(* IEC 61131-3 sources: AXOpen/src/components.rexroth.tightening/ctrl/src/Axo_CS351_compact (part 2) *)

                    Outputs.CwAnd := FALSE;
                    Outputs.CwLock := TRUE;

                    IF Inputs.CwLockAck THEN
                        THIS.CallTimers(FALSE);
                        _progress := 311;
                    END_IF;
                END_IF;
                // DisableClockwiseTask finished.
                IF _progress = 311 THEN
                    DisableClockwiseTask.DoneWhen(TRUE);
                    _progress := 0;
                END_IF;

                THIS.CallTimers(TRUE);

                DisableClockwiseTask.ThrowWhen(_errorTimer.output);
                Status.Action.Id := TO_UINT(_progress);
                DisableClockwiseTask.ThrowWhen(DisableClockwiseTask.Duration >= Config.TaskTimeout AND Config.TaskTimeout > T#0s ,'<#DisableClockwiseTask timeout.#>');
            END_IF;
            IF DisableClockwiseTask.DoneReached() THEN
                Status.Action.Id :=  UINT#111;
                Status.Error.Id :=  UINT#0;
            ELSIF DisableClockwiseTask.ErrorOccured() THEN
                Status.Action.Id :=  UINT#10010;
                Status.Error.Id  :=  UINT#10010;
            ELSIF DisableClockwiseTask.AbortTriggered()THEN
                Status.Action.Id :=  UINT#10011;
                Status.Error.Id  :=  UINT#10011;
            END_IF;
            Messenger.ActivateOnCondition(ULINT#10010,DisableClockwiseTask.HasError(), eAxoMessageCategory#Error);
            Messenger.ActivateOnCondition(ULINT#10011,DisableClockwiseTask.IsAborted(), eAxoMessageCategory#Error);
            Messenger.ActivateOnCondition(ULINT#112,DisableClockwiseTask.RestoreTriggered() , eAxoMessageCategory#Error);
            IF DisableClockwiseTask.RestoreTriggered() AND _progress >= 310 AND _progress <= 314  THEN
                Status.Action.Id :=  UINT#112;
                _progress := 0;
            END_IF;
            //**************************************************

            //*************EnableClockwiseTask******************
            EnableClockwiseTask.SetIsDisabled(FALSE);
            IF EnableClockwiseTask.StartTriggered() THEN
                Status.Action.Id :=  UINT#115;
            END_IF;
            Messenger.ActivateOnCondition(ULINT#115,EnableClockwiseTask.IsBusy(), eAxoMessageCategory#Info);
            Messenger.ActivateOnCondition(ULINT#116,EnableClockwiseTask.IsDone(), eAxoMessageCategory#Info);
            IF EnableClockwiseTask.Execute(THIS) THEN
                IF _progress = 0 THEN
                    Status.Error.Id := UINT#0;
                    TaskMessenger.Restore();
                    THIS.CallTimers(FALSE);
                    _progress := 315;
                END_IF;
                // EnableClockwiseTask running: waiting for 'Inputs.CwLockAck' to be off.
                IF _progress = 315 THEN
                    IF _infoTimer.output THEN
                        TaskMessenger.Activate( UINT#515, eAxoMessageCategory#Warning);
                        Status.Error.Id :=      UINT#515;
                    END_IF;

                    Outputs.CwAnd := TRUE;
                    Outputs.CwLock := FALSE;

                    IF NOT Inputs.CwLockAck THEN
                        THIS.CallTimers(FALSE);
                        _progress := 316;
                    END_IF;
                END_IF;
                // EnableClockwiseTask finished.
                IF _progress = 316 THEN
                    EnableClockwiseTask.DoneWhen(TRUE);
                    _progress := 0;
                END_IF;

                THIS.CallTimers(TRUE);

                EnableClockwiseTask.ThrowWhen(_errorTimer.output);
                Status.Action.Id := TO_UINT(_progress);
                EnableClockwiseTask.ThrowWhen(EnableClockwiseTask.Duration >= Config.TaskTimeout AND Config.TaskTimeout > T#0s ,'<#EnableClockwiseTask timeout.#>');
            END_IF;
            IF EnableClockwiseTask.DoneReached() THEN
                Status.Action.Id :=  UINT#116;
                Status.Error.Id :=  UINT#0;
            ELSIF EnableClockwiseTask.ErrorOccured() THEN
                Status.Action.Id :=  UINT#10015;
                Status.Error.Id  :=  UINT#10015;
            ELSIF EnableClockwiseTask.AbortTriggered()THEN
                Status.Action.Id :=  UINT#10016;
                Status.Error.Id  :=  UINT#10016;
            END_IF;
            Messenger.ActivateOnCondition(ULINT#10015,EnableClockwiseTask.HasError(), eAxoMessageCategory#Error);
            Messenger.ActivateOnCondition(ULINT#10016,EnableClockwiseTask.IsAborted(), eAxoMessageCategory#Error);
            Messenger.ActivateOnCondition(ULINT#117,EnableClockwiseTask.RestoreTriggered() , eAxoMessageCategory#Error);
            IF EnableClockwiseTask.RestoreTriggered() AND _progress >= 315 AND _progress <= 319  THEN
                Status.Action.Id :=  UINT#117;
                _progress := 0;
            END_IF;
            //**************************************************

            //*************DisableCounterClockwiseTask**********
            DisableCounterClockwiseTask.SetIsDisabled(FALSE);
            IF DisableCounterClockwiseTask.StartTriggered() THEN
                Status.Action.Id :=  UINT#120;
            END_IF;
            Messenger.ActivateOnCondition(ULINT#120,DisableCounterClockwiseTask.IsBusy(), eAxoMessageCategory#Info);
            Messenger.ActivateOnCondition(ULINT#121,DisableCounterClockwiseTask.IsDone(), eAxoMessageCategory#Info);
            IF DisableCounterClockwiseTask.Execute(THIS) THEN
                IF _progress = 0 THEN
                    Status.Error.Id := UINT#0;
                    TaskMessenger.Restore();
                    THIS.CallTimers(FALSE);
                    _progress := 320;
                END_IF;
                // DisableCounterClockwiseTask running: waiting for 'Inputs.CcwLockAck' to be on.
                IF _progress = 320 THEN
                    IF _infoTimer.output THEN
                        TaskMessenger.Activate( UINT#520, eAxoMessageCategory#Warning);
                        Status.Error.Id :=      UINT#520;
                    END_IF;

                    Outputs.CcwAnd := FALSE;
                    Outputs.CcwLock := TRUE;

                    IF Inputs.CcwLockAck THEN
                        THIS.CallTimers(FALSE);
                        _progress := 321;
                    END_IF;
                END_IF;
                // DisableCounterClockwiseTask  finished.
                IF _progress = 321 THEN
                    DisableCounterClockwiseTask.DoneWhen(TRUE);
                    _progress := 0;
                END_IF;

                THIS.CallTimers(TRUE);

                DisableCounterClockwiseTask.ThrowWhen(_errorTimer.output);
                Status.Action.Id := TO_UINT(_progress);
                DisableCounterClockwiseTask.ThrowWhen(DisableCounterClockwiseTask.Duration >= Config.TaskTimeout AND Config.TaskTimeout > T#0s ,'<#DisableCounterClockwiseTask timeout.#>');
            END_IF;
            IF DisableCounterClockwiseTask.DoneReached() THEN
                Status.Action.Id :=  UINT#121;
                Status.Error.Id :=  UINT#0;
            ELSIF DisableCounterClockwiseTask.ErrorOccured() THEN
                Status.Action.Id :=  UINT#10020;
                Status.Error.Id  :=  UINT#10020;
            ELSIF DisableCounterClockwiseTask.AbortTriggered()THEN
                Status.Action.Id :=  UINT#10021;
                Status.Error.Id  :=  UINT#10021;
            END_IF;
            Messenger.ActivateOnCondition(ULINT#10020,DisableCounterClockwiseTask.HasError(), eAxoMessageCategory#Error);
            Messenger.ActivateOnCondition(ULINT#10021,DisableCounterClockwiseTask.IsAborted(), eAxoMessageCategory#Error);
            Messenger.ActivateOnCondition(ULINT#122,DisableCounterClockwiseTask.RestoreTriggered() , eAxoMessageCategory#Error);
            IF DisableCounterClockwiseTask.RestoreTriggered() AND _progress >= 320 AND _progress <= 324  THEN
                Status.Action.Id :=  UINT#122;
                _progress := 0;
            END_IF;
            //**************************************************

            //*************EnableCounterClockwiseTask***********
            EnableCounterClockwiseTask.SetIsDisabled(FALSE);
            IF EnableCounterClockwiseTask.StartTriggered() THEN
                Status.Action.Id :=  UINT#125;
            END_IF;
            Messenger.ActivateOnCondition(ULINT#125,EnableCounterClockwiseTask.IsBusy(), eAxoMessageCategory#Info);
            Messenger.ActivateOnCondition(ULINT#126,EnableCounterClockwiseTask.IsDone(), eAxoMessageCategory#Info);
            IF EnableCounterClockwiseTask.Execute(THIS) THEN
                IF _progress = 0 THEN
                    Status.Error.Id := UINT#0;
                    TaskMessenger.Restore();
                    THIS.CallTimers(FALSE);
                    _progress := 325;
                END_IF;
                // EnableCounterClockwiseTask running: waiting for 'Inputs.CcwLockAck' to be off.
                IF _progress = 325 THEN
                    IF _infoTimer.output THEN
                        TaskMessenger.Activate( UINT#525, eAxoMessageCategory#Warning);
                        Status.Error.Id :=      UINT#525;
                    END_IF;

                    Outputs.CcwAnd := TRUE;
                    Outputs.CcwLock := FALSE;

                    IF NOT Inputs.CcwLockAck THEN
                        THIS.CallTimers(FALSE);
                        _progress := 326;
                    END_IF;
                END_IF;
                // EnableCounterClockwiseTask finished.
                IF _progress = 326 THEN
                    EnableCounterClockwiseTask.DoneWhen(TRUE);
                    _progress := 0;
                END_IF;

                THIS.CallTimers(TRUE);

                EnableCounterClockwiseTask.ThrowWhen(_errorTimer.output);
                Status.Action.Id := TO_UINT(_progress);
                EnableCounterClockwiseTask.ThrowWhen(EnableCounterClockwiseTask.Duration >= Config.TaskTimeout AND Config.TaskTimeout > T#0s ,'<#EnableCounterClockwiseTask timeout.#>');
            END_IF;
            IF EnableCounterClockwiseTask.DoneReached() THEN
                Status.Action.Id :=  UINT#126;
                Status.Error.Id :=  UINT#0;
            ELSIF EnableCounterClockwiseTask.ErrorOccured() THEN
                Status.Action.Id :=  UINT#10025;
                Status.Error.Id  :=  UINT#10025;
            ELSIF EnableCounterClockwiseTask.AbortTriggered()THEN
                Status.Action.Id :=  UINT#10026;
                Status.Error.Id  :=  UINT#10026;
            END_IF;
            Messenger.ActivateOnCondition(ULINT#10025,EnableCounterClockwiseTask.HasError(), eAxoMessageCategory#Error);
            Messenger.ActivateOnCondition(ULINT#10026,EnableCounterClockwiseTask.IsAborted(), eAxoMessageCategory#Error);
            Messenger.ActivateOnCondition(ULINT#127,EnableCounterClockwiseTask.RestoreTriggered() , eAxoMessageCategory#Error);
            IF EnableCounterClockwiseTask.RestoreTriggered() AND _progress >= 325 AND _progress <= 329  THEN
                Status.Action.Id :=  UINT#127;
                _progress := 0;
            END_IF;
            //**************************************************

            //*************ResetFaultTask***********************
            ResetFaultTask.SetIsDisabled(FALSE);
            IF ResetFaultTask.StartTriggered() THEN
                Status.Action.Id :=  UINT#130;
            END_IF;
            Messenger.ActivateOnCondition(ULINT#130,ResetFaultTask.IsBusy(), eAxoMessageCategory#Info);
            Messenger.ActivateOnCondition(ULINT#131,ResetFaultTask.IsDone(), eAxoMessageCategory#Info);
            IF ResetFaultTask.Execute(THIS) THEN
                IF _progress = 0 THEN
                    Status.Error.Id := UINT#0;
                    TaskMessenger.Restore();
                    THIS.CallTimers(FALSE);
                    _progress := 330;
                END_IF;
                // ResetFaultTask running: waiting for 'Inputs.NoFault' to be on.
                IF _progress = 330 THEN
                    IF _infoTimer.output THEN
                        TaskMessenger.Activate( UINT#530, eAxoMessageCategory#Warning);
                        Status.Error.Id :=      UINT#530;
                    END_IF;

                    Outputs.ResetFault := NOT Inputs.NoFault AND _blink.output;

                    IF Inputs.NoFault THEN
                        THIS.CallTimers(FALSE);
                        _progress := 331;
                    END_IF;
                END_IF;
                // ResetFaultTask running: waiting for 'Inputs.Ready' to be on.
                IF _progress = 331 THEN
                    IF _infoTimer.output THEN
                        TaskMessenger.Activate( UINT#531, eAxoMessageCategory#Warning);
                        Status.Error.Id :=      UINT#531;
                    END_IF;

                    IF Inputs.Ready THEN
                        THIS.CallTimers(FALSE);
                        _progress := 332;
                    END_IF;
                END_IF;
                // ResetFaultTask finished.
                IF _progress = 332 THEN
                    ResetFaultTask.DoneWhen(TRUE);
                    _progress := 0;
                END_IF;

                THIS.CallTimers(TRUE);

                ResetFaultTask.ThrowWhen(_errorTimer.output);
                Status.Action.Id := TO_UINT(_progress);
                ResetFaultTask.ThrowWhen(ResetFaultTask.Duration >= Config.TaskTimeout AND Config.TaskTimeout > T#0s ,'<#ResetFaultTask timeout.#>');
            END_IF;
            IF ResetFaultTask.DoneReached() THEN
                Status.Action.Id :=  UINT#131;
                Status.Error.Id :=  UINT#0;
            ELSIF ResetFaultTask.ErrorOccured() THEN
                Status.Action.Id :=  UINT#10030;
                Status.Error.Id  :=  UINT#10030;
            ELSIF ResetFaultTask.AbortTriggered()THEN
                Status.Action.Id :=  UINT#10031;
                Status.Error.Id  :=  UINT#10031;
            END_IF;
            Messenger.ActivateOnCondition(ULINT#10030,ResetFaultTask.HasError(), eAxoMessageCategory#Error);
            Messenger.ActivateOnCondition(ULINT#10031,ResetFaultTask.IsAborted(), eAxoMessageCategory#Error);
            Messenger.ActivateOnCondition(ULINT#132,ResetFaultTask.RestoreTriggered() , eAxoMessageCategory#Error);
            IF ResetFaultTask.RestoreTriggered() AND _progress >= 330 AND _progress <= 334  THEN
                Status.Action.Id :=  UINT#132;
                _progress := 0;
            END_IF;
            //**************************************************

            //*************ResetResultsTask*********************
            ResetResultsTask.SetIsDisabled(FALSE);
            IF ResetResultsTask.StartTriggered() THEN
                Status.Action.Id :=  UINT#135;
            END_IF;
            Messenger.ActivateOnCondition(ULINT#135,ResetResultsTask.IsBusy(), eAxoMessageCategory#Info);
            Messenger.ActivateOnCondition(ULINT#136,ResetResultsTask.IsDone(), eAxoMessageCategory#Info);
            IF ResetResultsTask.Execute(THIS) THEN
                IF _progress = 0 THEN
                    Status.Error.Id := UINT#0;
                    TaskMessenger.Restore();
                    THIS.CallTimers(FALSE);
                    _progress := 335;
                END_IF;
                // ResetResultsTask running: waiting for 'Inputs.CycleComplete' to be off.
                IF _progress = 335 THEN
                    IF _infoTimer.output THEN
                        TaskMessenger.Activate( UINT#535, eAxoMessageCategory#Warning);
                        Status.Error.Id :=      UINT#535;
                    END_IF;

                    Outputs.ResetResults := Inputs.CycleComplete AND _blink.output;
                    IF NOT Inputs.CycleComplete THEN
                        Outputs.ResetResults := FALSE;
                        THIS.CallTimers(FALSE);
                        _progress := 336;
                    END_IF;
                END_IF;
                // ResetResultsTask finished.
                IF _progress = 336 THEN
                    ResetResultsTask.DoneWhen(TRUE);
                    _progress := 0;
                END_IF;

                THIS.CallTimers(TRUE);

                ResetResultsTask.ThrowWhen(_errorTimer.output);
                Status.Action.Id := TO_UINT(_progress);
                ResetResultsTask.ThrowWhen(ResetResultsTask.Duration >= Config.TaskTimeout AND Config.TaskTimeout > T#0s ,'<#ResetResultsTask timeout.#>');
            END_IF;
            IF ResetResultsTask.DoneReached() THEN
                Status.Action.Id :=  UINT#136;
                Status.Error.Id :=  UINT#0;
            ELSIF ResetResultsTask.ErrorOccured() THEN
                Status.Action.Id :=  UINT#10035;
                Status.Error.Id  :=  UINT#10035;
            ELSIF ResetResultsTask.AbortTriggered()THEN
                Status.Action.Id :=  UINT#10036;
                Status.Error.Id  :=  UINT#10036;
            END_IF;
            Messenger.ActivateOnCondition(ULINT#10035,ResetResultsTask.HasError(), eAxoMessageCategory#Error);
            Messenger.ActivateOnCondition(ULINT#10036,ResetResultsTask.IsAborted(), eAxoMessageCategory#Error);
            Messenger.ActivateOnCondition(ULINT#137,ResetResultsTask.RestoreTriggered() , eAxoMessageCategory#Error);
            IF ResetResultsTask.RestoreTriggered() AND _progress >= 335 AND _progress <= 339  THEN
                Status.Action.Id :=  UINT#137;
                _progress := 0;
            END_IF;
            //**************************************************

            //*************SetScrewingProgramTask***************
            SetScrewingProgramTask.SetIsDisabled(FALSE);
            IF SetScrewingProgramTask.StartTriggered() THEN
                Status.Action.Id :=  UINT#140;
            END_IF;
            Messenger.ActivateOnCondition(ULINT#140,SetScrewingProgramTask.IsBusy(), eAxoMessageCategory#Info);
            Messenger.ActivateOnCondition(ULINT#141,SetScrewingProgramTask.IsDone(), eAxoMessageCategory#Info);
            IF SetScrewingProgramTask.Execute(THIS) THEN
                IF _progress = 0 THEN
                    Status.Error.Id := UINT#0;
                    TaskMessenger.Restore();
                    THIS.CallTimers(FALSE);
                    _progress := 340;
                END_IF;
                // SetScrewingProgramTask running: checking actual screwing program number.
                IF _progress = 340 THEN
                    IF _infoTimer.output THEN
                        TaskMessenger.Activate( UINT#540, eAxoMessageCategory#Warning);
                        Status.Error.Id :=      UINT#540;
                    END_IF;

                    IF _programNo <> Inputs.ProgramNo THEN
                        THIS.CallTimers(FALSE);
                        _progress := 341;
                    ELSE
                        THIS.CallTimers(FALSE);
                        _progress := 344;
                    END_IF;
                END_IF;
                // SetScrewingProgramTask running: checking required screwing program number.
                IF _progress = 341 THEN
                    IF _infoTimer.output THEN
                        TaskMessenger.Activate( UINT#541, eAxoMessageCategory#Warning);
                        Status.Error.Id :=      UINT#541;
                    END_IF;

                    IF _programNo>=BYTE#0 AND _programNo<=BYTE#99 THEN
                        THIS.CallTimers(FALSE);
                        _progress := 342;
                    ELSE
                        Messenger.Activate(ULINT#2000,eAxoMessageCategory#ProgrammingError);
                    END_IF;
                END_IF;
                // SetScrewingProgramTask running: waiting for 'Inputs.Ready' to be on.
                IF _progress = 342 THEN
                    IF _infoTimer.output THEN
                        TaskMessenger.Activate( UINT#542, eAxoMessageCategory#Warning);
                        Status.Error.Id :=      UINT#542;
                    END_IF;

                    IF Inputs.Ready THEN
                        THIS.CallTimers(FALSE);
                        _progress := 343;
                    END_IF;
                END_IF;
                // SetScrewingProgramTask running: waiting for the program to be set.
                IF _progress = 343 THEN
                    IF _infoTimer.output THEN
                        TaskMessenger.Activate( UINT#543, eAxoMessageCategory#Warning);
                        Status.Error.Id :=      UINT#543;
                    END_IF;

                    Outputs.ProgramNo := _programNo;

                    IF Inputs.ProgramNoAck = Outputs.ProgramNo THEN
                        THIS.CallTimers(FALSE);
                        _progress := 344;
                    END_IF;
                END_IF;
                // SetScrewingProgramTask finished.
                IF _progress = 344 THEN
                    SetScrewingProgramTask.DoneWhen(TRUE);
                    _progress := 0;
                END_IF;

                THIS.CallTimers(TRUE);

                SetScrewingProgramTask.ThrowWhen(_errorTimer.output);
                Status.Action.Id := TO_UINT(_progress);
                SetScrewingProgramTask.ThrowWhen(SetScrewingProgramTask.Duration >= Config.TaskTimeout AND Config.TaskTimeout > T#0s ,'<#SetScrewingProgramTask timeout.#>');
            END_IF;
            IF SetScrewingProgramTask.DoneReached() THEN
                Status.Action.Id :=  UINT#141;
                Status.Error.Id :=  UINT#0;
            ELSIF SetScrewingProgramTask.ErrorOccured() THEN
                Status.Action.Id :=  UINT#10040;
                Status.Error.Id  :=  UINT#10040;
            ELSIF SetScrewingProgramTask.AbortTriggered()THEN
                Status.Action.Id :=  UINT#10041;
                Status.Error.Id  :=  UINT#10041;
            END_IF;
            Messenger.ActivateOnCondition(ULINT#10040,SetScrewingProgramTask.HasError(), eAxoMessageCategory#Error);
            Messenger.ActivateOnCondition(ULINT#10041,SetScrewingProgramTask.IsAborted(), eAxoMessageCategory#Error);
            Messenger.ActivateOnCondition(ULINT#142,SetScrewingProgramTask.RestoreTriggered() , eAxoMessageCategory#Error);
            IF SetScrewingProgramTask.RestoreTriggered() AND _progress >= 340 AND _progress <= 344  THEN
                Status.Action.Id :=  UINT#142;
                _progress := 0;
            END_IF;
            //**************************************************

            //*************GetScrewingResultsTask*******************
            GetScrewingResultsTask.SetIsDisabled(FALSE);
            IF GetScrewingResultsTask.StartTriggered() THEN
                Status.Action.Id :=  UINT#150;
            END_IF;
            Messenger.ActivateOnCondition(ULINT#150,GetScrewingResultsTask.IsBusy(), eAxoMessageCategory#Info);
            Messenger.ActivateOnCondition(ULINT#151,GetScrewingResultsTask.IsDone(), eAxoMessageCategory#Info);
            IF GetScrewingResultsTask.Execute(THIS) THEN
                IF _progress = 0 THEN
                    Status.Error.Id := UINT#0;
                    TaskMessenger.Restore();
                    THIS.CallTimers(FALSE);
                    _progress := 350;
                END_IF;
                // GetScrewingResultsTask running.
                IF _progress = 350 THEN
                    IF _infoTimer.output THEN
                        TaskMessenger.Activate( UINT#550, eAxoMessageCategory#Warning);
                        Status.Error.Id :=      UINT#550;
                    END_IF;

                    Results.Result := Inputs.Result;
                    Results.IDcode.Data := Inputs.IDcode;
                    Results.CnoSE := Inputs.CnoSE;
                    Results.ProgramNo := Inputs.ProgramNo;
                    Results.TorqueMin := Inputs.TorqueMin;
                    Results.Torque := Inputs.Torque;
                    Results.TorqueMax := Inputs.TorqueMax;
                    Results.AngleMin := Inputs.AngleMin;
                    Results.Angle := Inputs.Angle;
                    Results.AngleMax := Inputs.AngleMax;
                    Results.ErrorCode := Inputs.ErrorCode;
                    Results.ErrorClass := Inputs.ErrorClass;

                    Results.IDcode.ToggleDataChangedFlag();

                    IF TRUE THEN
                        THIS.CallTimers(FALSE);
                        _progress := 351;
                    END_IF;
                END_IF;
                // GetScrewingResultsTask finished.
                IF _progress = 351 THEN
                    GetScrewingResultsTask.DoneWhen(TRUE);
                    _progress := 0;
                END_IF;

                THIS.CallTimers(TRUE);

                GetScrewingResultsTask.ThrowWhen(_errorTimer.output);
                Status.Action.Id := TO_UINT(_progress);
                GetScrewingResultsTask.ThrowWhen(GetScrewingResultsTask.Duration >= Config.TaskTimeout AND Config.TaskTimeout > T#0s ,'<#GetScrewingResultsTask timeout.#>');
            END_IF;
            IF GetScrewingResultsTask.DoneReached() THEN
                Status.Action.Id :=  UINT#151;
                Status.Error.Id :=  UINT#0;
            ELSIF GetScrewingResultsTask.ErrorOccured() THEN
                Status.Action.Id :=  UINT#10050;
                Status.Error.Id  :=  UINT#10050;
            ELSIF GetScrewingResultsTask.AbortTriggered()THEN
                Status.Action.Id :=  UINT#10051;
                Status.Error.Id  :=  UINT#10051;
            END_IF;
            Messenger.ActivateOnCondition(ULINT#10050,GetScrewingResultsTask.HasError(), eAxoMessageCategory#Error);
            Messenger.ActivateOnCondition(ULINT#10051,GetScrewingResultsTask.IsAborted(), eAxoMessageCategory#Error);
            Messenger.ActivateOnCondition(ULINT#152,GetScrewingResultsTask.RestoreTriggered() , eAxoMessageCategory#Error);
            IF GetScrewingResultsTask.RestoreTriggered() AND _progress >= 350 AND _progress <= 359  THEN
                Status.Action.Id :=  UINT#152;
                _progress := 0;
            END_IF;
            //**************************************************

            //*************ScrewClockwiseTask*******************
            ScrewClockwiseTask.SetIsDisabled(FALSE);
            IF ScrewClockwiseTask.StartTriggered() THEN
                Status.Action.Id :=  UINT#160;
            END_IF;
            Messenger.ActivateOnCondition(ULINT#160,ScrewClockwiseTask.IsBusy(), eAxoMessageCategory#Info);
            Messenger.ActivateOnCondition(ULINT#161,ScrewClockwiseTask.IsDone(), eAxoMessageCategory#Info);
            IF ScrewClockwiseTask.Execute(THIS) THEN
                IF _progress = 0 THEN
                    Status.Error.Id := UINT#0;
                    TaskMessenger.Restore();
                    THIS.CallTimers(FALSE);
                    _progress := 360;
                END_IF;
                // ScrewClockwiseTask running: waiting for 'Inputs.Ready' to be on.
                IF _progress = 360 THEN
                    IF _infoTimer.output THEN
                        TaskMessenger.Activate( UINT#560, eAxoMessageCategory#Warning);
                        Status.Error.Id :=      UINT#560;
                    END_IF;

                    IF Inputs.Ready THEN
                        THIS.CallTimers(FALSE);
                        _progress := 361;
                    END_IF;
                END_IF;
                // ScrewClockwiseTask running: waiting for 'Inputs.EnableAck' to be on.
                IF _progress = 361 THEN
                    IF _infoTimer.output THEN
                        TaskMessenger.Activate( UINT#561, eAxoMessageCategory#Warning);
                        Status.Error.Id :=      UINT#561;
                    END_IF;

                    Outputs.Enable := TRUE;
                    Outputs.ActiveEnable := TRUE;
                    IF Inputs.EnableAck THEN
                        THIS.CallTimers(FALSE);
                        _progress := 362;
                    END_IF;
                END_IF;
                // ScrewClockwiseTask running: waiting for 'Inputs.ActiveEnableAck' to be on.
                IF _progress = 362 THEN
                    IF _infoTimer.output THEN
                        TaskMessenger.Activate( UINT#562, eAxoMessageCategory#Warning);
                        Status.Error.Id :=      UINT#562;
                    END_IF;

                    Outputs.Enable := TRUE;
                    Outputs.ActiveEnable := TRUE;

                    IF Inputs.ActiveEnableAck THEN
                        THIS.CallTimers(FALSE);
                        _progress := 363;
                    END_IF;
                END_IF;
                // ScrewClockwiseTask running: waiting for 'Inputs.CwLockAck' to be off.
                IF _progress = 363 THEN
                    IF _infoTimer.output THEN
                        TaskMessenger.Activate( UINT#563, eAxoMessageCategory#Warning);
                        Status.Error.Id :=      UINT#563;
                    END_IF;

                    Outputs.CwAnd := TRUE;
                    Outputs.CwLock := FALSE;

                    IF NOT Inputs.CwLockAck THEN
                        THIS.CallTimers(FALSE);
                        _progress := 364;
                    END_IF;
                END_IF;
                // ScrewClockwiseTask running: waiting for 'Inputs.InCycle' to be on.
                IF _progress = 364 THEN
                    IF _infoTimer.output THEN
                        TaskMessenger.Activate( UINT#564, eAxoMessageCategory#Warning);
                        Status.Error.Id :=      UINT#564;
                    END_IF;

                    Outputs.StartClockwise := TRUE;

                    IF Inputs.InCycle THEN
                        THIS.CallTimers(FALSE);
                        _progress := 365;
                    END_IF;
                END_IF;
                // ScrewClockwiseTask running: waiting for 'Inputs.InCycle' to be on.
                IF _progress = 365 THEN
                    IF _infoTimer.output THEN
                        TaskMessenger.Activate( UINT#565, eAxoMessageCategory#Warning);
                        Status.Error.Id :=      UINT#565;
                    END_IF;

                    Outputs.StartClockwise := _automaticStart;

                    IF Inputs.InCycle THEN
                        THIS.CallTimers(FALSE);
                        _progress := 366;
                    END_IF;
                END_IF;
                // ScrewClockwiseTask running: waiting for 'Inputs.CycleComplete' to be on.
                IF _progress = 366 THEN
                    IF _infoTimer.output THEN
                        TaskMessenger.Activate( UINT#566, eAxoMessageCategory#Warning);
                        Status.Error.Id :=      UINT#566;
                    END_IF;

                    Outputs.StartClockwise := _automaticStart;

                    IF Inputs.CycleComplete THEN
                        THIS.CallTimers(FALSE);
                        _progress := 367;
                    END_IF;
                END_IF;
                // ScrewClockwiseTask running: waiting for 'Inputs.InCycle' to be off.
                IF _progress = 367 THEN
                    IF _infoTimer.output THEN
                        TaskMessenger.Activate( UINT#567, eAxoMessageCategory#Warning);
                        Status.Error.Id :=      UINT#567;
                    END_IF;

                    Outputs.StartClockwise := FALSE;
                    Outputs.ActiveEnable := FALSE;

                    IF NOT Inputs.InCycle THEN
                        THIS.CallTimers(FALSE);
                        _progress := 368;
                    END_IF;
                END_IF;
                // ScrewClockwiseTask running: waiting for 'Inputs.ActiveEnableAck' to be off.
                IF _progress = 368 THEN
                    IF _infoTimer.output THEN
                        TaskMessenger.Activate( UINT#568, eAxoMessageCategory#Warning);
                        Status.Error.Id :=      UINT#568;
                    END_IF;

                    Outputs.StartClockwise := FALSE;
                    Outputs.ActiveEnable := FALSE;

                    IF NOT Inputs.ActiveEnableAck THEN
                        THIS.CallTimers(FALSE);
                        _progress := 369;
                    END_IF;
                END_IF;
                // ScrewClockwiseTask running: waiting for 'Inputs.CycleComplete' to be on.
                IF _progress = 369 THEN
                    IF _infoTimer.output THEN
                        TaskMessenger.Activate( UINT#569, eAxoMessageCategory#Warning);
                        Status.Error.Id :=      UINT#569;
                    END_IF;

                    Outputs.StartClockwise := FALSE;
                    Outputs.ActiveEnable := FALSE;

                    IF Inputs.CycleComplete THEN
                        THIS.CallTimers(FALSE);
                        _progress := 370;
                    END_IF;
                END_IF;
                // ScrewClockwiseTask running: waiting for 'Inputs.CwLockAck' to be on.
                IF _progress = 370 THEN
                    IF _infoTimer.output THEN
                        TaskMessenger.Activate( UINT#570, eAxoMessageCategory#Warning);
                        Status.Error.Id :=      UINT#570;
                    END_IF;

                    Outputs.CwAnd := FALSE;
                    Outputs.CwLock := TRUE;

                    IF Inputs.CwLockAck THEN
                        THIS.CallTimers(FALSE);
                        _progress := 371;
                    END_IF;
                END_IF;
                // ScrewClockwiseTask running: waiting for 'Inputs.CcwLockAck' to be on.
                IF _progress = 371 THEN
                    IF _infoTimer.output THEN
                        TaskMessenger.Activate( UINT#571, eAxoMessageCategory#Warning);
                        Status.Error.Id :=      UINT#571;
                    END_IF;

                    Outputs.CcwAnd := FALSE;
                    Outputs.CcwLock := TRUE;

                   IF Inputs.CcwLockAck THEN
                        THIS.CallTimers(FALSE);
                        _progress := 372;
                    END_IF;
                END_IF;
                // ScrewClockwiseTask finished.
                IF _progress = 372 THEN
                    ScrewClockwiseTask.DoneWhen(TRUE);
                    _progress := 0;
                END_IF;

                THIS.CallTimers(TRUE);

                ScrewClockwiseTask.ThrowWhen(_errorTimer.output);
                Status.Action.Id := TO_UINT(_progress);
                ScrewClockwiseTask.ThrowWhen(ScrewClockwiseTask.Duration >= Config.TaskTimeout AND Config.TaskTimeout > T#0s ,'<#ScrewClockwiseTask timeout.#>');
            END_IF;
            IF ScrewClockwiseTask.DoneReached() THEN
                Status.Action.Id :=  UINT#161;
                Status.Error.Id :=  UINT#0;
            ELSIF ScrewClockwiseTask.ErrorOccured() THEN
                Status.Action.Id :=  UINT#10060;
                Status.Error.Id  :=  UINT#10060;
            ELSIF ScrewClockwiseTask.AbortTriggered()THEN
                Status.Action.Id :=  UINT#10061;
                Status.Error.Id  :=  UINT#10061;
            END_IF;
            Messenger.ActivateOnCondition(ULINT#10060,ScrewClockwiseTask.HasError(), eAxoMessageCategory#Error);
            Messenger.ActivateOnCondition(ULINT#10061,ScrewClockwiseTask.IsAborted(), eAxoMessageCategory#Error);
            Messenger.ActivateOnCondition(ULINT#162,ScrewClockwiseTask.RestoreTriggered() , eAxoMessageCategory#Error);
            IF ScrewClockwiseTask.RestoreTriggered() AND _progress >= 360 AND _progress <= 379  THEN
                Status.Action.Id :=  UINT#162;
                _progress := 0;
            END_IF;
            //*****************************************************

            //*************ScrewCounterClockwiseTask***************
            ScrewCounterClockwiseTask.SetIsDisabled(FALSE);
            IF ScrewCounterClockwiseTask.StartTriggered() THEN
                Status.Action.Id :=  UINT#180;
            END_IF;
            Messenger.ActivateOnCondition(ULINT#180,ScrewCounterClockwiseTask.IsBusy(), eAxoMessageCategory#Info);
            Messenger.ActivateOnCondition(ULINT#181,ScrewCounterClockwiseTask.IsDone(), eAxoMessageCategory#Info);
            IF ScrewCounterClockwiseTask.Execute(THIS) THEN
                IF _progress = 0 THEN
                    Status.Error.Id := UINT#0;
                    TaskMessenger.Restore();
                    THIS.CallTimers(FALSE);
                    _progress := 380;
                END_IF;
                // ScrewCounterClockwiseTask running: waiting for 'Inputs.Ready' to be on.
                IF _progress = 380 THEN
                    IF _infoTimer.output THEN
                        TaskMessenger.Activate( UINT#580, eAxoMessageCategory#Warning);
                        Status.Error.Id :=      UINT#580;
                    END_IF;

                    IF Inputs.Ready THEN
                        THIS.CallTimers(FALSE);
                        _progress := 381;
                    END_IF;
                END_IF;
                // ScrewCounterClockwiseTask running: waiting for 'Inputs.EnableAck' to be on.
                IF _progress = 381 THEN
                    IF _infoTimer.output THEN
                        TaskMessenger.Activate( UINT#581, eAxoMessageCategory#Warning);
                        Status.Error.Id :=      UINT#581;
                    END_IF;

                    Outputs.Enable := TRUE;
                    Outputs.ActiveEnable := TRUE;
                    IF Inputs.EnableAck THEN
                        THIS.CallTimers(FALSE);
                        _progress := 382;
                    END_IF;
                END_IF;
                // ScrewCounterClockwiseTask running: waiting for 'Inputs.ActiveEnableAck' to be on.
                IF _progress = 382 THEN
                    IF _infoTimer.output THEN
                        TaskMessenger.Activate( UINT#582, eAxoMessageCategory#Warning);
                        Status.Error.Id :=      UINT#582;
                    END_IF;

                    Outputs.Enable := TRUE;
                    Outputs.ActiveEnable := TRUE;
                    IF Inputs.ActiveEnableAck THEN
                        THIS.CallTimers(FALSE);
                        _progress := 383;
                    END_IF;
                END_IF;
                // ScrewCounterClockwiseTask running: waiting for 'Inputs.CcwLockAck' to be off.
                IF _progress = 383 THEN
                    IF _infoTimer.output THEN
                        TaskMessenger.Activate( UINT#583, eAxoMessageCategory#Warning);
                        Status.Error.Id :=      UINT#583;
                    END_IF;

                    Outputs.CcwAnd := TRUE;
                    Outputs.CcwLock := FALSE;
                    IF NOT Inputs.CcwLockAck THEN
                        THIS.CallTimers(FALSE);
                        _progress := 384;
                    END_IF;
                END_IF;
                // ScrewCounterClockwiseTask running: waiting for 'Inputs.InCycleCcw' to be on.
                IF _progress = 384 THEN
                    IF _infoTimer.output THEN
                        TaskMessenger.Activate( UINT#584, eAxoMessageCategory#Warning);
                        Status.Error.Id :=      UINT#584;
                    END_IF;

                    IF _automaticStart THEN
                        Outputs.StartCounterClockwise := TRUE;
                    END_IF;
                    IF Inputs.InCycleCcw THEN
                        THIS.CallTimers(FALSE);
                        _progress := 385;
                    END_IF;
                END_IF;
                // ScrewCounterClockwiseTask running: waiting for 'Inputs.InCycleCcw' to be on.
                IF _progress = 385 THEN
                    IF _infoTimer.output THEN
                        TaskMessenger.Activate( UINT#585, eAxoMessageCategory#Warning);
                        Status.Error.Id :=      UINT#585;
                    END_IF;

                    Outputs.StartCounterClockwise := TRUE;
                    IF Inputs.InCycleCcw THEN
                        THIS.CallTimers(FALSE);
                        _progress := 386;
                    END_IF;
                END_IF;
                // ScrewCounterClockwiseTask running: waiting for 'Inputs.CycleComplete' to be on.
                IF _progress = 386 THEN
                    IF _infoTimer.output THEN
                        TaskMessenger.Activate( UINT#586, eAxoMessageCategory#Warning);
                        Status.Error.Id :=      UINT#586;
                    END_IF;

                    Outputs.StartCounterClockwise := TRUE;
                    IF Inputs.CycleComplete THEN
                        THIS.CallTimers(FALSE);
                        _progress := 387;
                    END_IF;
                END_IF;
                // ScrewCounterClockwiseTask running: waiting for 'Inputs.InCycleCcw' to be off.
                IF _progress = 387 THEN
                    IF _infoTimer.output THEN
                        TaskMessenger.Activate( UINT#587, eAxoMessageCategory#Warning);
                        Status.Error.Id :=      UINT#587;
                    END_IF;

                    Outputs.StartCounterClockwise := FALSE;
                    Outputs.ActiveEnable := FALSE;

                    IF NOT Inputs.InCycleCcw THEN
                        THIS.CallTimers(FALSE);
                        _progress := 388;
                    END_IF;
                END_IF;
                // ScrewCounterClockwiseTask running: waiting for 'Inputs.ActiveEnableAck' to be off.
                IF _progress = 388 THEN
                    IF _infoTimer.output THEN
                        TaskMessenger.Activate( UINT#588, eAxoMessageCategory#Warning);
                        Status.Error.Id :=      UINT#588;
                    END_IF;

                    Outputs.StartCounterClockwise := FALSE;
                    Outputs.ActiveEnable := FALSE;

                    IF NOT Inputs.ActiveEnableAck THEN
                        THIS.CallTimers(FALSE);
                        _progress := 389;
                    END_IF;
                END_IF;
                // ScrewCounterClockwiseTask running: waiting for 'Inputs.CycleComplete' to be on.
                IF _progress = 389 THEN
                    IF _infoTimer.output THEN
                        TaskMessenger.Activate( UINT#589, eAxoMessageCategory#Warning);
                        Status.Error.Id :=      UINT#589;
                    END_IF;

                    Outputs.StartCounterClockwise := FALSE;
                    Outputs.ActiveEnable := FALSE;

                    IF Inputs.CycleComplete THEN
                        THIS.CallTimers(FALSE);
                        _progress := 390;
                    END_IF;
                END_IF;
                // ScrewCounterClockwiseTask running: waiting for 'Inputs.CcwLockAck' to be on.
                IF _progress = 390 THEN
                    IF _infoTimer.output THEN
                        TaskMessenger.Activate( UINT#590, eAxoMessageCategory#Warning);
                        Status.Error.Id :=      UINT#590;
                    END_IF;

                    Outputs.CcwAnd := FALSE;
                    Outputs.CcwLock := TRUE;
                    IF Inputs.CcwLockAck THEN
                        THIS.CallTimers(FALSE);
                        _progress := 391;
                    END_IF;
                END_IF;
                // ScrewCounterClockwiseTask running: waiting for 'Inputs.CwLockAck' to be on.
                IF _progress = 391 THEN
                    IF _infoTimer.output THEN
                        TaskMessenger.Activate( UINT#591, eAxoMessageCategory#Warning);
                        Status.Error.Id :=      UINT#591;
                    END_IF;

                    Outputs.CwAnd := FALSE;
                    Outputs.CwLock := TRUE;
                    IF Inputs.CwLockAck THEN
                        THIS.CallTimers(FALSE);
                        _progress := 392;
                    END_IF;
                END_IF;
                // ScrewCounterClockwiseTask finished.
                IF _progress = 392 THEN
                    ScrewCounterClockwiseTask.DoneWhen(TRUE);
                    _progress := 0;
                END_IF;

                THIS.CallTimers(TRUE);

                ScrewCounterClockwiseTask.ThrowWhen(_errorTimer.output);
                Status.Action.Id := TO_UINT(_progress);
                ScrewCounterClockwiseTask.ThrowWhen(ScrewCounterClockwiseTask.Duration >= Config.TaskTimeout AND Config.TaskTimeout > T#0s ,'<#ScrewCounterClockwiseTask timeout.#>');
            END_IF;
            IF ScrewCounterClockwiseTask.DoneReached() THEN
                Status.Action.Id :=  UINT#181;
                Status.Error.Id :=  UINT#0;
            ELSIF ScrewCounterClockwiseTask.ErrorOccured() THEN
                Status.Action.Id :=  UINT#10080;
                Status.Error.Id  :=  UINT#10080;
            ELSIF ScrewCounterClockwiseTask.AbortTriggered()THEN
                Status.Action.Id :=  UINT#10081;
                Status.Error.Id  :=  UINT#10081;
            END_IF;
            Messenger.ActivateOnCondition(ULINT#10080,ScrewCounterClockwiseTask.HasError(), eAxoMessageCategory#Error);
            Messenger.ActivateOnCondition(ULINT#10081,ScrewCounterClockwiseTask.IsAborted(), eAxoMessageCategory#Error);
            Messenger.ActivateOnCondition(ULINT#182,ScrewCounterClockwiseTask.RestoreTriggered() , eAxoMessageCategory#Error);
            IF ScrewCounterClockwiseTask.RestoreTriggered() AND _progress >= 380 AND _progress <= 399  THEN
                Status.Action.Id :=  UINT#182;
                _progress := 0;
            END_IF;
            //**************************************************

            //*************RunAutomatTask***********************
            RunAutomatTask.SetIsDisabled(FALSE);
            IF RunAutomatTask.StartTriggered() THEN
                Status.Action.Id :=  UINT#200;
            END_IF;
            Messenger.ActivateOnCondition(ULINT#200,RunAutomatTask.IsBusy(), eAxoMessageCategory#Info);
            Messenger.ActivateOnCondition(ULINT#201,RunAutomatTask.IsDone(), eAxoMessageCategory#Info);
            IF RunAutomatTask.Execute(THIS) THEN
                IF _progress = 0 THEN
                    Status.Error.Id := UINT#0;
                    TaskMessenger.Restore();
                    THIS.CallTimers(FALSE);
                    _progress := 400;
                END_IF;
                // RunAutomatTask running: setting ID code.
                IF _progress = 400 THEN
                    IF _infoTimer.output THEN
                        TaskMessenger.Activate( UINT#600, eAxoMessageCategory#Warning);
                        Status.Error.Id :=      UINT#600;
                    END_IF;

                    OK := FALSE;
                    NOK := FALSE;

                    Outputs.IDcode := _IDcode;

                    IF TRUE THEN
                        THIS.CallTimers(FALSE);
                        _progress := 401;
                    END_IF;
                END_IF;
                // RunAutomatTask running: waiting for 'Inputs.NoFault' to be on.
                IF _progress = 401 THEN
                    IF _infoTimer.output THEN
                        TaskMessenger.Activate( UINT#601, eAxoMessageCategory#Warning);
                        Status.Error.Id :=      UINT#601;
                    END_IF;

                    Outputs.ResetFault := NOT Inputs.NoFault AND _blink.output;
                    IF Inputs.NoFault THEN
                        Outputs.ResetFault := FALSE;
                        THIS.CallTimers(FALSE);
                        _progress := 402;
                    END_IF;
                END_IF;
                // RunAutomatTask running: waiting for 'Inputs.Ready' to be on.
                IF _progress = 402 THEN
                    IF _infoTimer.output THEN
                        TaskMessenger.Activate( UINT#602, eAxoMessageCategory#Warning);
                        Status.Error.Id :=      UINT#602;
                    END_IF;

                    Outputs.ResetFault := NOT Inputs.NoFault AND _blink.output;
                    IF Inputs.Ready THEN
                        Outputs.ResetFault := FALSE;
                        THIS.CallTimers(FALSE);
                        _progress := 403;
                    END_IF;
                END_IF;
                // RunAutomatTask running: checking the actual screwing program number.
                IF _progress = 403 THEN
                    IF _infoTimer.output THEN
                        TaskMessenger.Activate( UINT#603, eAxoMessageCategory#Warning);
                        Status.Error.Id :=      UINT#603;
                    END_IF;

                    IF _programNo <> Inputs.ProgramNo THEN
                        THIS.CallTimers(FALSE);
                        _progress := 404;
                    ELSE
                        THIS.CallTimers(FALSE);
                        _progress := 407;
                    END_IF;
                END_IF;
                // RunAutomatTask running: checking the required screwing program number
                IF _progress = 404 THEN
                    IF _infoTimer.output THEN
                        TaskMessenger.Activate( UINT#604, eAxoMessageCategory#Warning);
                        Status.Error.Id :=      UINT#604;
                    END_IF;

                    IF _programNo>=BYTE#0 AND _programNo<=BYTE#99 THEN
                        THIS.CallTimers(FALSE);
                        _progress := 405;
                    ELSE
                        Messenger.Activate(ULINT#1100,eAxoMessageCategory#ProgrammingError);
                    END_IF;
                END_IF;
                // RunAutomatTask running: waiting for 'Inputs.Ready' to be on.
                IF _progress = 405 THEN
                    IF _infoTimer.output THEN
                        TaskMessenger.Activate( UINT#605, eAxoMessageCategory#Warning);
                        Status.Error.Id :=      UINT#605;
                    END_IF;

                    IF Inputs.Ready THEN
                        THIS.CallTimers(FALSE);
                        _progress := 406;
                    END_IF;
                END_IF;
                // RunAutomatTask running: waiting for the screwing program to be set.
                IF _progress = 406 THEN
                    IF _infoTimer.output THEN
                        TaskMessenger.Activate( UINT#606, eAxoMessageCategory#Warning);
                        Status.Error.Id :=      UINT#606;
                    END_IF;

                    Outputs.ProgramNo := _programNo;

                    IF Inputs.ProgramNoAck = Outputs.ProgramNo THEN
                        THIS.CallTimers(FALSE);
                        _progress := 407;
                    END_IF;
                END_IF;
                // RunAutomatTask running: waiting for 'Inputs.EnableAck' to be on.
                IF _progress = 407 THEN
                    IF _infoTimer.output THEN
                        TaskMessenger.Activate( UINT#607, eAxoMessageCategory#Warning);
                        Status.Error.Id :=      UINT#607;
                    END_IF;

                    Outputs.Enable := TRUE;

                    IF Inputs.EnableAck THEN
                        THIS.CallTimers(FALSE);
                        _progress := 408;
                    END_IF;
                END_IF;
                // RunAutomatTask running: waiting for 'Inputs.CycleComplete' to be off.
                IF _progress = 408 THEN
                    IF _infoTimer.output THEN
                        TaskMessenger.Activate( UINT#608, eAxoMessageCategory#Warning);
                        Status.Error.Id :=      UINT#608;
                    END_IF;

                    Outputs.ResetResults := Inputs.CycleComplete AND _blink.output;
                    IF NOT Inputs.CycleComplete THEN
                        Outputs.ResetResults := FALSE;
                        THIS.CallTimers(FALSE);
                        _progress := 409;
                    END_IF;
                END_IF;
                // RunAutomatTask running: waiting for 'Inputs.ActiveEnableAck' to be on.
                IF _progress = 409 THEN
                    IF _infoTimer.output THEN
                        TaskMessenger.Activate( UINT#609, eAxoMessageCategory#Warning);
                        Status.Error.Id :=      UINT#609;
                    END_IF;

                    Outputs.ActiveEnable := TRUE;
                    IF Inputs.ActiveEnableAck THEN
                        THIS.CallTimers(FALSE);
                        _progress := 410;
                    END_IF;
                END_IF;
                // RunAutomatTask running: waiting for 'Inputs.CwLockAck' to be off.
                IF _progress = 410 THEN
                    IF _infoTimer.output THEN
                        TaskMessenger.Activate( UINT#610, eAxoMessageCategory#Warning);
                        Status.Error.Id :=      UINT#610;
                    END_IF;

                    Outputs.CwAnd := TRUE;
                    Outputs.CwLock := FALSE;
                    IF NOT Inputs.CwLockAck THEN
                        THIS.CallTimers(FALSE);
                        _progress := 411;
                    END_IF;
                END_IF;
                // RunAutomatTask running: waiting for 'Inputs.InCycle' to be on.
                IF _progress = 411 THEN
                    IF _infoTimer.output THEN
                        TaskMessenger.Activate( UINT#611, eAxoMessageCategory#Warning);
                        Status.Error.Id :=      UINT#611;
                    END_IF;

                    Outputs.StartClockwise := TRUE;
                    IF Inputs.InCycle THEN
                        THIS.CallTimers(FALSE);
                        _progress := 412;
                    END_IF;
                END_IF;
                // RunAutomatTask running: waiting for 'Inputs.InCycle' to be on.
                IF _progress = 412 THEN
                    IF _infoTimer.output THEN
                        TaskMessenger.Activate( UINT#612, eAxoMessageCategory#Warning);
                        Status.Error.Id :=      UINT#612;
                    END_IF;

                    IF _automaticStart THEN
                        Outputs.StartClockwise := TRUE;
                    END_IF;
                    IF Inputs.InCycle THEN
                        THIS.CallTimers(FALSE);
                        _progress := 413;
                    END_IF;
                END_IF;
                // RunAutomatTask running: waiting for 'Inputs.CycleComplete' to be on.
                IF _progress = 413 THEN
                    IF _infoTimer.output THEN
                        TaskMessenger.Activate( UINT#613, eAxoMessageCategory#Warning);
                        Status.Error.Id :=      UINT#613;
                    END_IF;

                    IF _automaticStart THEN
                        Outputs.StartClockwise := TRUE;
                    END_IF;
                    IF Inputs.CycleComplete THEN
                        THIS.CallTimers(FALSE);
                        _progress := 414;
                    END_IF;
                END_IF;
                // RunAutomatTask running: waiting for 'Inputs.InCycle' to be off.
                IF _progress = 414 THEN
                    IF _infoTimer.output THEN
                        TaskMessenger.Activate( UINT#614, eAxoMessageCategory#Warning);
                        Status.Error.Id :=      UINT#614;
                    END_IF;

                    Outputs.StartClockwise := FALSE;
                    Outputs.ActiveEnable := FALSE;
                    IF NOT Inputs.InCycle THEN
                        THIS.CallTimers(FALSE);
                        _progress := 415;
                    END_IF;
                END_IF;
                // RunAutomatTask running: waiting for 'Inputs.ActiveEnableAck' to be off.
                IF _progress = 415 THEN
                    IF _infoTimer.output THEN
                        TaskMessenger.Activate( UINT#615, eAxoMessageCategory#Warning);
                        Status.Error.Id :=      UINT#615;
                    END_IF;

                    Outputs.StartClockwise := FALSE;
                    Outputs.ActiveEnable := FALSE;

                    IF NOT Inputs.ActiveEnableAck THEN
                        THIS.CallTimers(FALSE);
                        _progress := 416;
                    END_IF;
                END_IF;
                // RunAutomatTask running: waiting for 'Inputs.CycleComplete' to be on.
                IF _progress = 416 THEN
                    IF _infoTimer.output THEN
                        TaskMessenger.Activate( UINT#616, eAxoMessageCategory#Warning);
                        Status.Error.Id :=      UINT#616;
                    END_IF;

                    Outputs.StartClockwise := FALSE;
                    Outputs.ActiveEnable := FALSE;

                    IF Inputs.CycleComplete THEN
                        THIS.CallTimers(FALSE);
                        _progress := 417;
                    END_IF;
                END_IF;
                // RunAutomatTask running: waiting for 'Inputs.CwLockAck' to be on.
                IF _progress = 417 THEN
                    IF _infoTimer.output THEN
                        TaskMessenger.Activate( UINT#617, eAxoMessageCategory#Warning);
                        Status.Error.Id :=      UINT#617;
                    END_IF;

                    Outputs.CwAnd := FALSE;
                    Outputs.CwLock := TRUE;

                    IF Inputs.CwLockAck THEN
                        THIS.CallTimers(FALSE);
                        _progress := 418;
                    END_IF;
                END_IF;
                // RunAutomatTask running: waiting for 'Inputs.CcwLockAck' to be on.
                IF _progress = 418 THEN
                    IF _infoTimer.output THEN
                        TaskMessenger.Activate( UINT#618, eAxoMessageCategory#Warning);
                        Status.Error.Id :=      UINT#618;
                    END_IF;

                    Outputs.CcwAnd := FALSE;
                    Outputs.CcwLock := TRUE;

                    IF Inputs.CcwLockAck THEN
                        THIS.CallTimers(FALSE);
                        _progress := 419;
                    END_IF;
                END_IF;
                // RunAutomatTask running: saving screwing results.
                IF _progress = 419 THEN
                    IF _infoTimer.output THEN
                        TaskMessenger.Activate( UINT#619, eAxoMessageCategory#Warning);
                        Status.Error.Id :=      UINT#619;
                    END_IF;

                    Results.Result := Inputs.Result;
                    Results.IDcode.Data := Inputs.IDcode;
                    Results.CnoSE := Inputs.CnoSE;
                    Results.ProgramNo := Inputs.ProgramNo;
                    Results.TorqueMin := Inputs.TorqueMin;
                    Results.Torque := Inputs.Torque;
                    Results.TorqueMax := Inputs.TorqueMax;
                    Results.AngleMin := Inputs.AngleMin;
                    Results.Angle := Inputs.Angle;
                    Results.AngleMax := Inputs.AngleMax;
                    Results.ErrorCode := Inputs.ErrorCode;
                    Results.ErrorClass := Inputs.ErrorClass;

                    Results.IDcode.ToggleDataChangedFlag();

                    IF TRUE THEN
                        THIS.CallTimers(FALSE);
                        _progress := 420;
                    END_IF;
                END_IF;
                // RunAutomatTask running: evaluating screwing results.
                IF _progress = 420 THEN
                    IF _infoTimer.output THEN
                        TaskMessenger.Activate( UINT#620, eAxoMessageCategory#Warning);
                        Status.Error.Id :=      UINT#620;
                    END_IF;

                    OK := Inputs.OK AND NOT Inputs.NOK;
                    NOK := NOT Inputs.OK OR Inputs.NOK;
                    IF OK OR NOK THEN
                        THIS.CallTimers(FALSE);
                        _progress := 421;
                    END_IF;
                END_IF;
                // RunAutomatTask running: waiting for 'Inputs.EnableAck' to be off.
                IF _progress = 421 THEN
                    IF _infoTimer.output THEN
                        TaskMessenger.Activate( UINT#621, eAxoMessageCategory#Warning);
                        Status.Error.Id :=      UINT#621;
                    END_IF;

                    Outputs.Enable := FALSE;

                    IF NOT Inputs.EnableAck THEN
                        THIS.CallTimers(FALSE);
                        _progress := 422;
                    END_IF;
                END_IF;
                // RunAutomatTask finished.
                IF _progress = 422 THEN
                    RunAutomatTask.DoneWhen(TRUE);
                    _progress := 0;
                END_IF;

                THIS.CallTimers(TRUE);

                RunAutomatTask.ThrowWhen(_errorTimer.output);
                Status.Action.Id := TO_UINT(_progress);
                RunAutomatTask.ThrowWhen(RunAutomatTask.Duration >= Config.TaskTimeout AND Config.TaskTimeout > T#0s ,'<#RunAutomatTask timeout.#>');
            END_IF;
            IF RunAutomatTask.DoneReached() THEN
                Status.Action.Id :=  UINT#201;
                Status.Error.Id :=  UINT#0;
            ELSIF RunAutomatTask.ErrorOccured() THEN
                Status.Action.Id :=  UINT#10100;
                Status.Error.Id  :=  UINT#10100;
            ELSIF RunAutomatTask.AbortTriggered()THEN
                Status.Action.Id :=  UINT#10101;
                Status.Error.Id  :=  UINT#10101;
            END_IF;
            Messenger.ActivateOnCondition(ULINT#10100,RunAutomatTask.HasError(), eAxoMessageCategory#Error);
            Messenger.ActivateOnCondition(ULINT#10101,RunAutomatTask.IsAborted(), eAxoMessageCategory#Error);
            Messenger.ActivateOnCondition(ULINT#202,RunAutomatTask.RestoreTriggered() , eAxoMessageCategory#Error);
            IF RunAutomatTask.RestoreTriggered() AND _progress >= 400 AND _progress <= 439  THEN
                Status.Action.Id :=  UINT#202;
                _progress := 0;
            END_IF;
            //**************************************************

            //***********Update outputs ****************
            // Slot 1 Output_4_word_1
            _data_out4w[0].%B1        :=      Outputs.ProgramNo;                      //  0

            _data_out4w[0].%X0        :=      Outputs.Enable;                         //  1
            _data_out4w[0].%X1        :=      Outputs.ResetFault;
            _data_out4w[0].%X2        :=      Outputs.StartClockwise;
            _data_out4w[0].%X3        :=      Outputs.StartCounterClockwise;
            _data_out4w[0].%X4        :=      Outputs.ResetResults;
            _data_out4w[0].%X5        :=      Outputs.NokAck;
            _data_out4w[0].%X6        :=      Outputs.UsrIn1;
            _data_out4w[0].%X7        :=      Outputs.UsrIn2;

            _data_out4w[1].%X8        :=      Outputs.ES_LED_Green;                   //  2
            _data_out4w[1].%X9        :=      Outputs.ES_LED_Yellow;
            _data_out4w[1].%X10       :=      Outputs.ES_LED_Red;
            _data_out4w[1].%X11       :=      Outputs.ActiveEnable;
            _data_out4w[1].%X12       :=      Outputs.CcwLock;
            _data_out4w[1].%X13       :=      Outputs.CwLock;
            _data_out4w[1].%X14       :=      Outputs.CwAnd;
            _data_out4w[1].%X15       :=      Outputs.CcwAnd;

            _data_out4w[2].%B1        :=      Outputs.IDcode[0];                      //  4
            _data_out4w[2].%B0        :=      Outputs.IDcode[1];                      //  5
            _data_out4w[3].%B1        :=      Outputs.IDcode[2];                      //  6
            _data_out4w[3].%B0        :=      Outputs.IDcode[3];                      //  7

            _returnValue := Siemens.Simatic.DistributedIO.WriteData((Config.HWIDs.HwID_Slot_1),_data_out4w);
            IF _returnValue > WORD#0 THEN
                Messenger.Activate(UINT#1231, eAxoMessageCategory#Error);
                Status.Error.Id := UINT#1231;
                RETURN;
            END_IF;

            // Slot 2 Output_4_word_2
            _data_out4w[0].%B1        :=      Outputs.IDcode[4];                      //  8
            _data_out4w[0].%B0        :=      Outputs.IDcode[5];                      //  9
            _data_out4w[1].%B1        :=      Outputs.IDcode[6];                      //  10
            _data_out4w[1].%B0        :=      Outputs.IDcode[7];                      //  11
            _data_out4w[2].%B1        :=      Outputs.IDcode[8];                      //  12
            _data_out4w[2].%B0        :=      Outputs.IDcode[9];                      //  13
            _data_out4w[3].%B1        :=      Outputs.IDcode[10];                     //  14
            _data_out4w[3].%B0        :=      Outputs.IDcode[11];                     //  15

            _returnValue := Siemens.Simatic.DistributedIO.WriteData((Config.HWIDs.HwID_Slot_2),_data_out4w);
            IF _returnValue > WORD#0 THEN
                Messenger.Activate(UINT#1232, eAxoMessageCategory#Error);
                Status.Error.Id := UINT#1232;
                RETURN;
            END_IF;

            // Slot 3 Output_4_word_3
            _data_out4w[0].%B1        :=      Outputs.IDcode[12];                     //  16
            _data_out4w[0].%B0        :=      Outputs.IDcode[13];                     //  17
            _data_out4w[1].%B1        :=      Outputs.IDcode[14];                     //  18
            _data_out4w[1].%B0        :=      Outputs.IDcode[15];                     //  19
            _data_out4w[2].%B1        :=      Outputs.IDcode[16];                     //  20
            _data_out4w[2].%B0        :=      Outputs.IDcode[17];                     //  21
            _data_out4w[3].%B1        :=      Outputs.IDcode[18];                     //  22
            _data_out4w[3].%B0        :=      Outputs.IDcode[19];                     //  23

            _returnValue := Siemens.Simatic.DistributedIO.WriteData((Config.HWIDs.HwID_Slot_3),_data_out4w);
            IF _returnValue > WORD#0 THEN
                Messenger.Activate(UINT#1233, eAxoMessageCategory#Error);
                Status.Error.Id := UINT#1233;
                RETURN;
            END_IF;

            // Slot 4 Output_4_word_4
            _data_out4w[0].%B1        :=      Outputs.IDcode[20];                     //  24
            _data_out4w[0].%B0        :=      Outputs.IDcode[21];                     //  25
            _data_out4w[1].%B1        :=      Outputs.IDcode[22];                     //  26
            _data_out4w[1].%B0        :=      Outputs.IDcode[23];                     //  27
            _data_out4w[2].%B1        :=      Outputs.IDcode[24];                     //  28
            _data_out4w[2].%B0        :=      Outputs.IDcode[25];                     //  29
            _data_out4w[3].%B1        :=      Outputs.IDcode[26];                     //  30
            _data_out4w[3].%B0        :=      Outputs.IDcode[27];                     //  31

            _returnValue := Siemens.Simatic.DistributedIO.WriteData((Config.HWIDs.HwID_Slot_4),_data_out4w);
            IF _returnValue > WORD#0 THEN
                Messenger.Activate(UINT#1234, eAxoMessageCategory#Error);
                Status.Error.Id := UINT#1234;
                RETURN;
            END_IF;

            // Slot 5 Output_4_word_5
            _data_out4w[0].%B1        :=      Outputs.IDcode[28];                     //  32
            _data_out4w[0].%B0        :=      Outputs.IDcode[29];                     //  33
            _data_out4w[1].%B1        :=      Outputs.IDcode[30];                     //  34
            _data_out4w[1].%B0        :=      Outputs.IDcode[31];                     //  35
            _data_out4w[2].%B1        :=      Outputs.IDcode[32];                     //  36
            _data_out4w[2].%B0        :=      Outputs.IDcode[33];                     //  37
            _data_out4w[3].%B1        :=      Outputs.IDcode[34];                     //  38
            _data_out4w[3].%B0        :=      Outputs.IDcode[35];                     //  39

            _returnValue := Siemens.Simatic.DistributedIO.WriteData((Config.HWIDs.HwID_Slot_5),_data_out4w);
            IF _returnValue > WORD#0 THEN
                Messenger.Activate(UINT#1235, eAxoMessageCategory#Error);
                Status.Error.Id := UINT#1235;
                RETURN;
            END_IF;

            // Slot 6 Output_4_word_6
            _data_out4w[0].%B1        :=      Outputs.IDcode[36];                     //  40
            _data_out4w[0].%B0        :=      Outputs.IDcode[37];                     //  41
            _data_out4w[1].%B1        :=      Outputs.IDcode[38];                     //  42
            _data_out4w[1].%B0        :=      Outputs.IDcode[39];                     //  43
            _data_out4w[2].%B1        :=      Outputs.IDcode[40];                     //  44
            _data_out4w[2].%B0        :=      Outputs.IDcode[41];                     //  45
            _data_out4w[3].%B1        :=      Outputs.IDcode[42];                     //  46
            _data_out4w[3].%B0        :=      Outputs.IDcode[43];                     //  47

            _returnValue := Siemens.Simatic.DistributedIO.WriteData((Config.HWIDs.HwID_Slot_6),_data_out4w);
            IF _returnValue > WORD#0 THEN
                Messenger.Activate(UINT#1236, eAxoMessageCategory#Error);
                Status.Error.Id := UINT#1236;
                RETURN;
            END_IF;

            // Slot 7 Output_4_word_7
            _data_out4w[0].%B1        :=      Outputs.IDcode[44];                     //  48
            _data_out4w[0].%B0        :=      Outputs.IDcode[45];                     //  49
            _data_out4w[1].%B1        :=      Outputs.IDcode[46];                     //  50
            _data_out4w[1].%B0        :=      Outputs.IDcode[47];                     //  51
            _data_out4w[2].%B1        :=      Outputs.IDcode[48];                     //  52
            _data_out4w[2].%B0        :=      Outputs.IDcode[49];                     //  53
            _data_out4w[3].%B1        :=      Outputs.IDcode[50];                     //  54
            _data_out4w[3].%B0        :=      Outputs.IDcode[51];                     //  55

            _returnValue := Siemens.Simatic.DistributedIO.WriteData((Config.HWIDs.HwID_Slot_7),_data_out4w);
            IF _returnValue > WORD#0 THEN
                Messenger.Activate(UINT#1237, eAxoMessageCategory#Error);
                Status.Error.Id := UINT#1237;
                RETURN;
            END_IF;

            // Slot 8 Output_4_word_8
            _data_out4w[0].%B1        :=      Outputs.IDcode[52];                     //  56
            _data_out4w[0].%B0        :=      Outputs.IDcode[53];                     //  57
            _data_out4w[1].%B1        :=      Outputs.IDcode[54];                     //  58
            _data_out4w[1].%B0        :=      Outputs.IDcode[55];                     //  59
            _data_out4w[2].%B1        :=      Outputs.IDcode[56];                     //  60
            _data_out4w[2].%B0        :=      Outputs.IDcode[57];                     //  61
            _data_out4w[3].%B1        :=      Outputs.IDcode[58];                     //  62
            _data_out4w[3].%B0        :=      Outputs.IDcode[59];                     //  63

            _returnValue := Siemens.Simatic.DistributedIO.WriteData((Config.HWIDs.HwID_Slot_8),_data_out4w);
            IF _returnValue > WORD#0 THEN
                Messenger.Activate(UINT#1238, eAxoMessageCategory#Error);
                Status.Error.Id := UINT#1238;
                RETURN;
            END_IF;

            // Slot 9 Output_2_word_1
            _data_out2w[0].%B1        :=      Outputs.IDcode[60];                     //  64
            _data_out2w[0].%B0        :=      Outputs.IDcode[61];                     //  65
            _data_out2w[1].%B1        :=      Outputs.IDcode[62];                     //  66
            _data_out2w[1].%B0        :=      Outputs.IDcode[63];                     //  67

            _returnValue := Siemens.Simatic.DistributedIO.WriteData((Config.HWIDs.HwID_Slot_9),_data_out2w);
            IF _returnValue > WORD#0 THEN
                Messenger.Activate(UINT#1239, eAxoMessageCategory#Error);
                Status.Error.Id := UINT#1239;
                RETURN;
            END_IF;
            //******************************************

        END_METHOD

        METHOD PUBLIC Disable : IAxoTaskState
            Disable := DisableTask.Invoke(THIS);
        END_METHOD

        METHOD PUBLIC Enable : IAxoTaskState
            Enable := EnableTask.Invoke(THIS);
        END_METHOD

        METHOD PUBLIC DisableClockwise : IAxoTaskState
            DisableClockwise := DisableClockwiseTask.Invoke(THIS);
        END_METHOD

        METHOD PUBLIC EnableClockwise : IAxoTaskState
            EnableClockwise := EnableClockwiseTask.Invoke(THIS);
        END_METHOD

        METHOD PUBLIC DisableCounterClockwise : IAxoTaskState
            DisableCounterClockwise := DisableCounterClockwiseTask.Invoke(THIS);
        END_METHOD

        METHOD PUBLIC EnableCounterClockwise : IAxoTaskState
            EnableCounterClockwise := EnableCounterClockwiseTask.Invoke(THIS);
        END_METHOD

        METHOD PUBLIC ResetFault : IAxoTaskState
            ResetFault := ResetFaultTask.Invoke(THIS);
        END_METHOD

        METHOD PUBLIC ResetResults : IAxoTaskState
            ResetResults := ResetResultsTask.Invoke(THIS);
        END_METHOD

        METHOD PUBLIC SetScrewingProgram : IAxoTaskState
            VAR_INPUT
                ProgramNo : BYTE;
            END_VAR
            _programNo  :=  ProgramNo;
            SetScrewingProgram := SetScrewingProgramTask.Invoke(THIS);
        END_METHOD

        METHOD PUBLIC GetScrewingResults : IAxoTaskState
            GetScrewingResults := GetScrewingResultsTask.Invoke(THIS);
        END_METHOD

        METHOD PUBLIC ScrewClockwise : IAxoTaskState
            VAR_INPUT
                AutomaticStart : BOOL;
            END_VAR
            _automaticStart := AutomaticStart;
            ScrewClockwise := ScrewClockwiseTask.Invoke(THIS);
        END_METHOD

        METHOD PUBLIC ScrewCounterClockwise : IAxoTaskState
            VAR_INPUT
                AutomaticStart : BOOL;
            END_VAR
            _automaticStart := AutomaticStart;
            ScrewCounterClockwise := ScrewCounterClockwiseTask.Invoke(THIS);
        END_METHOD

        METHOD PUBLIC RunAutomat : IAxoTaskState
            VAR_INPUT
                ProgramNo : BYTE;
                IDcode : STRING[64];
                AutomaticStart : BOOL;
            END_VAR
            VAR
               _data : ARRAY[0..64] OF BYTE;
               _i   :   UINT;
            END_VAR
            Serialize(UDINT#0, IDcode, _data);
            _programNo  :=  ProgramNo;
            FOR _i := UINT#1 TO UINT#64 DO
                _IDcode[_i - UINT#1] := _data[_i];
            END_FOR;
            _automaticStart := AutomaticStart;
            RunAutomat := RunAutomatTask.Invoke(THIS);
        END_METHOD

        METHOD PROTECTED OVERRIDE ManualControl
            VAR
                _data : ARRAY[0..64] OF BYTE;
                _i   :   UINT;
             END_VAR
             Serialize(UDINT#0, IDcodeManual, _data);
             _programNo  :=  ProgramNoManual;
             FOR _i := UINT#1 TO UINT#64 DO
                 _IDcode[_i - UINT#1] := _data[_i];
             END_FOR;
             _automaticStart := AutomaticStartManual;
            THIS._isManuallyControllable := TRUE;
        END_METHOD

        ///<summary>
        /// Restores this component into intial state.
        ///</summary>
        METHOD PUBLIC OVERRIDE Restore
            VAR
                _index : INT;
            END_VAR
            Status.Action.Id := UINT#0;
            Status.Error.Id  := UINT#0;

            _progress       :=   INT#0;
            _returnValue    :=   WORD#0;

            _data_in4w[0] := WORD#0;
            _data_in4w[1] := WORD#0;
            _data_in4w[2] := WORD#0;
            _data_in4w[3] := WORD#0;

            _data_out4w[0] := WORD#0;
            _data_out4w[1] := WORD#0;
            _data_out4w[2] := WORD#0;
            _data_out4w[3] := WORD#0;

            _data_out2w[0] := WORD#0;
            _data_out2w[1] := WORD#0;

            _word           :=   WORD#0;
            _dword          :=   DWORD#0;

            DisableTask.Restore();
            EnableTask.Restore();
            DisableClockwiseTask.Restore();
            EnableClockwiseTask.Restore();
            DisableCounterClockwiseTask.Restore();
            EnableCounterClockwiseTask.Restore();
            ResetFaultTask.Restore();
            ResetResultsTask.Restore();
            SetScrewingProgramTask.Restore();
            GetScrewingResultsTask.Restore();

            ScrewClockwiseTask.Restore();
            ScrewCounterClockwiseTask.Restore();
            RunAutomatTask.Restore();
            HardwareDiagnosticsTask.Restore();

            Status.Action.Id := UINT#50;
            RestoreTask.DoneWhen(TRUE);

        END_METHOD

        METHOD PRIVATE CallTimers
            VAR_INPUT
                signal : BOOL;
            END_VAR

            _infoTimer.OnDelay(THIS, signal AND Config.InfoTime > LT#0S ,Config.InfoTime);
            _errorTimer.OnDelay(THIS, signal AND Config.ErrorTime > LT#0S , Config.ErrorTime);
        END_METHOD
    END_CLASS
END_NAMESPACE
